INTERFACE I_AteqComm

METHOD M_Update : BOOL
VAR_INPUT
END_VAR
END_METHOD

END_INTERFACE

(* stored: Version 1.1.0.1, ProductVersion 3.1.4024.15
   Itf I_AteqComm: Id {71c1248e-87e1-4e4d-a330-3120d5fe4056}
   Method M_Update: Id {45feac3a-d2d1-44bf-a0ca-7f7d0f81e6ca} *)
